Universal Robots URScript: test.script

def test():
  global _hidden_verificationVariable=0
  set_target_payload(0.260000, [0.050000, -0.008000, 0.024000], [0.000163, 0.000163, 0.000163, 0.000000, 0.000000, 0.000000])
  set_tool_communication(False, 115200, 0, 1, 1.5, 3.5)
  set_tool_output_mode(0)
  set_tool_digital_output_mode(0, 1)
  set_tool_digital_output_mode(1, 1)
  set_tool_voltage(0)
  set_safety_mode_transition_hardness(1)
  set_tcp(p[0.028210348281514253,-0.09610723587300697,-0.09969041498611403,0.0,0.0,0.0])
  set_gravity([0.0, 0.0, 9.82])
  set_standard_analog_input_domain(0, 1)
  set_standard_analog_input_domain(1, 1)
  set_tool_analog_input_domain(0, 1)
  set_tool_analog_input_domain(1, 1)
  set_analog_outputdomain(0, 0)
  set_analog_outputdomain(1, 0)
  set_input_actions_to_default()
  global Plane_1=p[0.32571614183608727,0.7933870146316717,0.11820742021636722,-2.208244884171713,-0.24738609815952348,-1.9195085473101943]
  global Plane_2=p[0.3436052139151623,0.7478032414335104,0.10077839665899768,2.768545736097797,0.1284831553507919,1.3672805628273381]
  global Plane_3=p[0.31945151854627996,0.6757990361168175,0.09459088830114093,2.7301760593116526,-0.049483824131046385,1.4252239353300047]
  global Plane_4=p[0.3372257363094211,0.6222230974198586,0.07001667903587716,2.621672423508307,-0.12240385890263918,1.4373011913128484]
  # begin: URCap Installation Node
  #   Source: External Control, 1.0.5, FZI Research Center for Information Technology
  #   Type: External Control
  # end: URCap Installation Node
  step_count_d25caf92_c5d0_4b0d_8346_bd69edc4ae2a = 0.0
  thread Step_Counter_Thread_6b3826c6_650f_4c6e_ac5b_63da6eb62561():
    while (True):
      step_count_d25caf92_c5d0_4b0d_8346_bd69edc4ae2a = step_count_d25caf92_c5d0_4b0d_8346_bd69edc4ae2a + 1.0
      sync()
    end
  end
  run Step_Counter_Thread_6b3826c6_650f_4c6e_ac5b_63da6eb62561()
  global Waypoint_5_p=p[.331961491069, .722321069848, .108294054993, -1.644924239511, -2.108127402866, 1.059041005191]
  global Waypoint_5_q=[-2.263827625659779, -0.3747088467210835, 0.9072378304888372, -1.3311374645588119, -1.3414838949653225, -2.600121562840531]
  global Waypoint_1_p=p[.338919302833, .665001489926, .114260142464, -1.637779241863, -2.114844316195, 1.080412956872]
  global Waypoint_1_q=[-2.318634812031852, -0.4877417844585352, 1.1314995924579938, -1.4215563547662775, -1.3917120138751216, -2.643481318150635]
  global Waypoint_4_p=p[.338919302833, .665001489926, .114260142464, -1.637779241863, -2.114844316195, 1.080412956872]
  global Waypoint_4_q=[-2.318634812031852, -0.4877417844585352, 1.1314995924579938, -1.4215563547662775, -1.3917120138751216, -2.643481318150635]
  global Waypoint_2_p=p[.331961491088, .722321069696, .108294055009, -1.644924241075, -2.108127401663, 1.059041006074]
  global Waypoint_2_q=[-2.263827625905569, -0.3747088474198179, 0.9072378317708427, -1.3311374646915493, -1.3414838949729022, -2.600121561666377]
  def d_eighth():
    $ 5 "d_eighth" "noBreak"
    $ 6 "MoveL"
    $ 7 "Waypoint_5" "breakAfter"
    movel(pose_trans(Plane_2, pose_trans(p[-.360194635270, .718115715874, -.204939404457, -2.768545736098, -.128483155351, -1.367280562827], Waypoint_5_p)), a=1.2, v=0.25)
    $ 8 "Waypoint_1" "breakAfter"
    movel(pose_trans(Plane_2, pose_trans(p[-.360194635270, .718115715874, -.204939404457, -2.768545736098, -.128483155351, -1.367280562827], Waypoint_1_p)), a=1.2, v=0.25)
  end
  def d_eighthUp():
    $ 9 "d_eighthUp" "noBreak"
    $ 10 "MoveL"
    $ 11 "Waypoint_4" "breakAfter"
    movel(pose_trans(Plane_2, pose_trans(p[-.360194635270, .718115715874, -.204939404457, -2.768545736098, -.128483155351, -1.367280562827], Waypoint_4_p)), a=1.2, v=0.25)
    $ 12 "Waypoint_2" "breakAfter"
    movel(pose_trans(Plane_2, pose_trans(p[-.360194635270, .718115715874, -.204939404457, -2.768545736098, -.128483155351, -1.367280562827], Waypoint_2_p)), a=1.2, v=0.25)
  end
  $ 2 "Robot Program"
  $ 3 "Call d_eighth"
  d_eighth()
  $ 4 "Call d_eighthUp"
  d_eighthUp()
end
